{attribute addProperty BoxType "AT2050-0501-0020"}
{attribute addProperty Id "A_0087_AT2050_5501_0016_AT2050_5501AT2050_C5E5984862678.25"}
{attribute addProperty CRC "1804001523"}
{attribute addProperty SizeInBites "626"}
{attribute addProperty SizeInBytes "78.25"}
TYPE A_0057_AT2050_0501_0020_6B86E0F3 EXTENDS AT2050_BA5A9548 :
STRUCT
	{attribute addProperty Name "A_0087_AT2050_5501_0016_AT2050_5501"}
	A_0087_AT2050_5501_0016_AT2050_5501 : AT2050_C5E59848;
END_STRUCT
END_TYPE

(* stored: Version 1.2.0.0, ProductVersion 3.1.4024.9
   DUT A_0057_AT2050_0501_0020_6B86E0F3: Id {035eeded-cf2e-4767-9daa-edd7c8bd0392} *)
